FUNCTION_BLOCK FB_Ampel
VAR_INPUT
	eState : BOOL;
END_VAR
VAR_OUTPUT
	bAmpelGruen : BOOL;
	bAmpelRot : BOOL;
	bAmpelGelb : BOOL;
END_VAR
VAR
END_VAR

END_FUNCTION_BLOCK

(* stored: Version 1.1.0.1, ProductVersion 3.1.4024.15
   POU FB_Ampel: Id {d9081e82-d3cf-4285-9890-cb1a91f12aff}, SpecialFunc None *)
